// TIA Portal V16 export
// export: Created 2021-07-12T14:47:19.4773321Z, ExportSetting WithDefaults, DisplayName Totally Integrated Automation Portal, DisplayVersion V16, DisplayName TIA Portal Version Control Interface, DisplayVersion V16, DisplayName TIA Portal Openness, DisplayVersion V16, DisplayName STEP 7 Professional, DisplayVersion V16, DisplayName STEP 7 Safety, DisplayVersion V16, DisplayName WinCC Professional, DisplayVersion V16
TYPE "LSimaHydTO_typeActorDirectionValves"
TITLE = LSimaHydTO_typeActorDirectionValves
// Settings of the direction valves control
// stored: IsFailsafeCompliant false
   STRUCT
      WaitTimeByDirectionChange { S7_SetPoint := 'True'} : LReal := 0.0;   // Waiting time between switching the digital valve valveForward and valveBackward for a direction change [s]
      DelayTimeValveForward { S7_SetPoint := 'True'} : LReal := 0.0;   // Reaction time for digital valve [s]
      DelayTimeValveBackward { S7_SetPoint := 'True'} : LReal := 0.0;   // Reaction time for digital valve [s]
      ValvesOffMode { S7_SetPoint := 'True'} : DInt := 0;   // 0: keep digital valves on after ramp down / 1: switch off digital valves after ramp down
      DisplacementForce { S7_SetPoint := 'True'} : Bool := FALSE;   // 1: force control by displacement ( inverse direction), e.g. die cushion
   END_STRUCT;
END_TYPE
